% RSLogix 500 project Hourmeter.RSS, saved by version 8.30.00.16 %
PROJECT "SIM_PLC"    % processor: Bul.1763 MicroLogix 1100 Series B %

PROGRAM FILES
  LAD 2 "MAIN"  3 rungs
  LAD 3 "INPUTS"  3 rungs
  LAD 4 "CTRL LOGIC"  8 rungs

DATA FILES
  O0 OUTPUT  4 elements
  I1 INPUT  7 elements
  S2 STATUS  66 elements
  B3 BINARY  1 elements
  T4 TIMER  1 elements
  C5 COUNTER  4 elements
  R6 CONTROL  1 elements
  N7 INTEGER  4 elements
  F8 FLOAT  1 elements

LADDER 2 "MAIN"
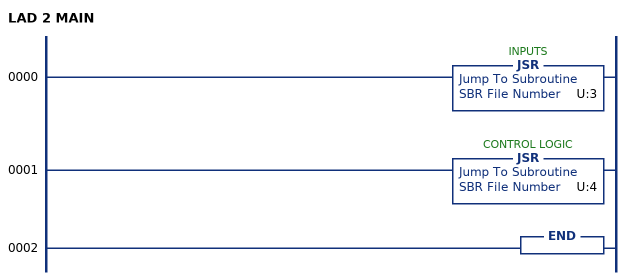
% Rung: 0 %
SOR JSR U:3 EOR
%   U:3  "INPUTS" %
% Rung: 1 %
SOR JSR U:4 EOR
%   U:4  "CONTROL LOGIC" %
% Rung: 2 %
SOR END EOR

LADDER 3 "INPUTS"
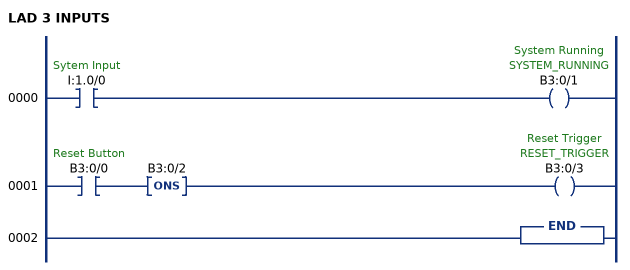
% Rung: 0 %
SOR XIC I:1.0/0 OTE B3:0/1 EOR
%   I:1.0/0  "Sytem Input" %
%   B3:0/1  SYSTEM_RUNNING  "System Running" %
% Rung: 1 %
SOR XIC B3:0/0 ONS B3:0/2 OTE B3:0/3 EOR
%   B3:0/0  "Reset Button" %
%   B3:0/3  RESET_TRIGGER  "Reset Trigger" %
% Rung: 2 %
SOR END EOR

LADDER 4 "CTRL LOGIC"
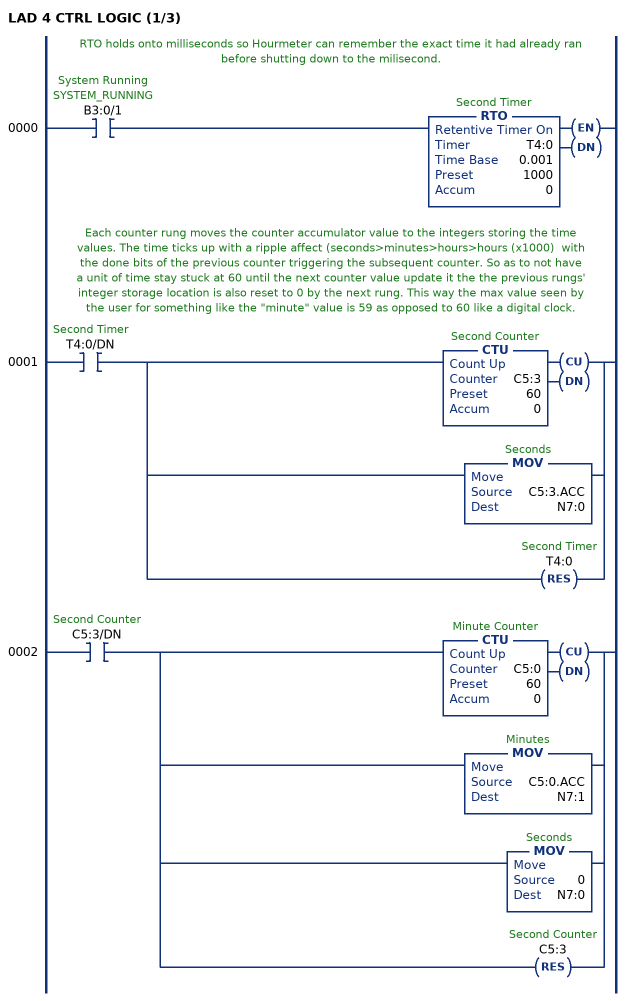
% Rung: 0 %
% RTO holds onto milliseconds so Hourmeter can remember the exact time it had already ran before shutting down to the milisecond. %
SOR XIC B3:0/1 RTO T4:0 0.001 1000 0 EOR
%   B3:0/1  SYSTEM_RUNNING  "System Running" %
%   T4:0  "Second Timer" %
% Rung: 1 %  % edit flag set %
% Each counter rung moves the counter accumulator value to the integers storing the time values. The time ticks up with a ripple affect (seconds>minutes>hours>hours (x1000)  with the done bits of the previous counter triggering the subsequent counter. So as to not have a unit of time stay stuck at 60 until the next counter value update it the the previous rungs' integer storage location is also reset to 0 by the next rung. This way the max value seen by the user for something like the "minute" value is 59 as opposed to 60 like a digital clock. %
SOR XIC T4:0/DN BST CTU C5:3 60 0 NXB MOV C5:3.ACC N7:0 NXB RES T4:0 BND EOR
%   T4:0  "Second Timer" %
%   C5:3  "Second Counter" %
%   N7:0  "Seconds" %
% Rung: 2 %
SOR XIC C5:3/DN BST CTU C5:0 60 0 NXB MOV C5:0.ACC N7:1 NXB MOV 0 N7:0 NXB RES C5:3 BND EOR
%   C5:3  "Second Counter" %
%   C5:0  "Minute Counter" %
%   N7:1  "Minutes" %
%   N7:0  "Seconds" %

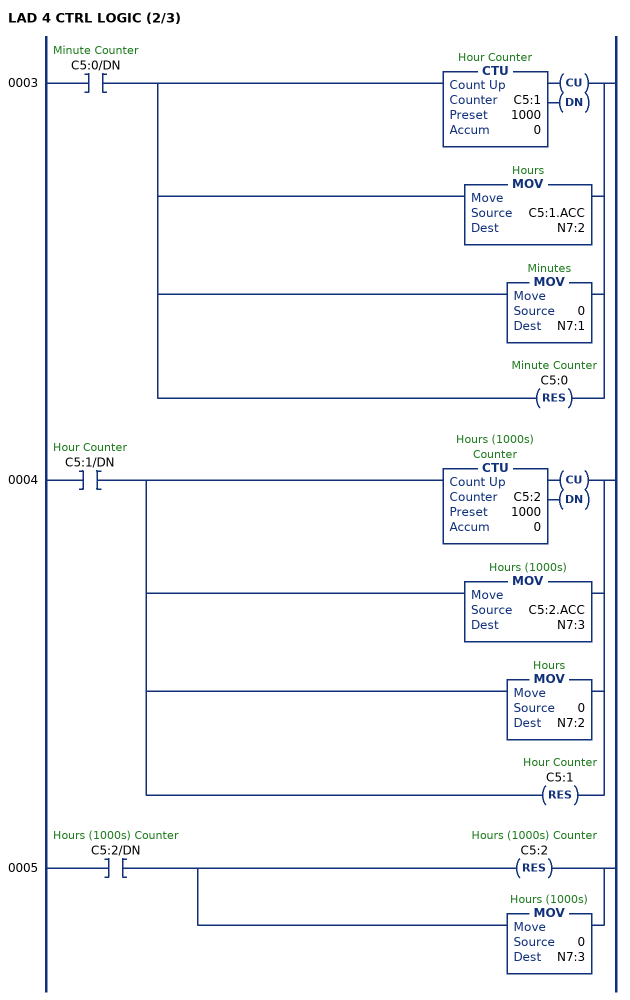
% Rung: 3 %
SOR XIC C5:0/DN BST CTU C5:1 1000 0 NXB MOV C5:1.ACC N7:2 NXB MOV 0 N7:1 NXB RES C5:0 BND EOR
%   C5:0  "Minute Counter" %
%   C5:1  "Hour Counter" %
%   N7:2  "Hours" %
%   N7:1  "Minutes" %
% Rung: 4 %
SOR XIC C5:1/DN BST CTU C5:2 1000 0 NXB MOV C5:2.ACC N7:3 NXB MOV 0 N7:2 NXB RES C5:1 BND EOR
%   C5:1  "Hour Counter" %
%   C5:2  "Hours (1000s) Counter" %
%   N7:3  "Hours (1000s)" %
%   N7:2  "Hours" %
% Rung: 5 %
SOR XIC C5:2/DN BST RES C5:2 NXB MOV 0 N7:3 BND EOR
%   C5:2  "Hours (1000s) Counter" %
%   N7:3  "Hours (1000s)" %

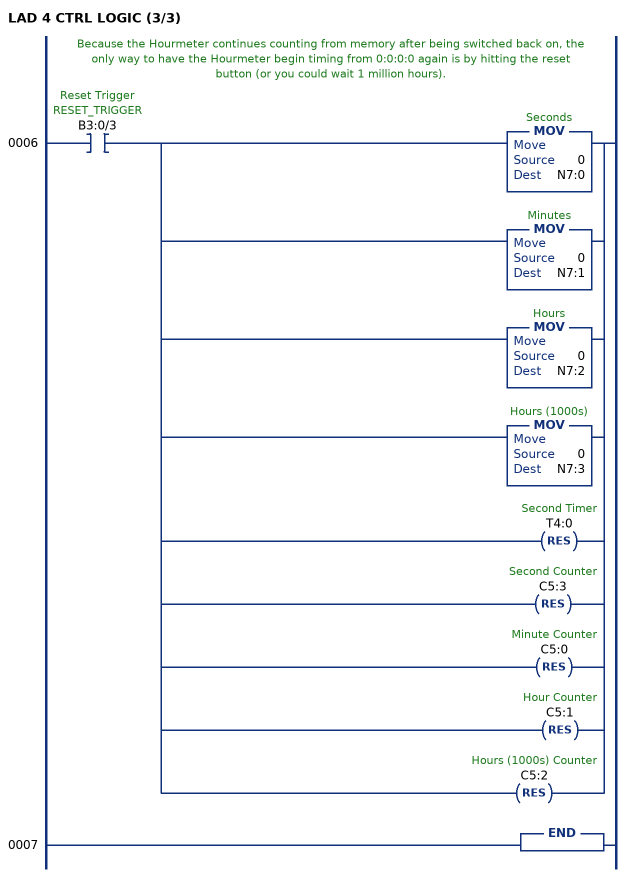
% Rung: 6 %
% Because the Hourmeter continues counting from memory after being switched back on, the only way to have the Hourmeter begin timing from 0:0:0:0 again is by hitting the reset button (or you could wait 1 million hours). %
SOR XIC B3:0/3 BST MOV 0 N7:0 NXB MOV 0 N7:1 NXB MOV 0 N7:2 NXB MOV 0 N7:3 NXB RES T4:0 NXB RES C5:3 NXB RES C5:0 NXB RES C5:1 NXB RES C5:2 BND EOR
%   B3:0/3  RESET_TRIGGER  "Reset Trigger" %
%   N7:0  "Seconds" %
%   N7:1  "Minutes" %
%   N7:2  "Hours" %
%   N7:3  "Hours (1000s)" %
%   T4:0  "Second Timer" %
%   C5:3  "Second Counter" %
%   C5:0  "Minute Counter" %
%   C5:1  "Hour Counter" %
%   C5:2  "Hours (1000s) Counter" %
% Rung: 7 %
SOR END EOR

COMMENTS NOT ATTACHED TO A CURRENT RUNG
  T4:0: RTO holds onto milliseconds so Hourmeter can remember the exact time it had already ran before shutting down to the milisecond.

DATA TABLE (non-zero values as saved)
DATA T4
% .PRE .ACC %
% T4:0 % 1000 0
DATA C5
% .PRE .ACC %
% C5:0 % 60 0
% C5:1 % 1000 0
% C5:2 % 1000 0
% C5:3 % 60 0
